FUNCTION_BLOCK GR_plant_Without_NDT
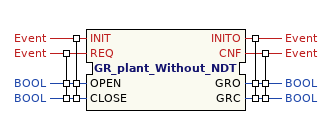
  EVENT_INPUT
    INIT WITH OPEN, CLOSE;
    REQ WITH OPEN, CLOSE;
  END_EVENT
  EVENT_OUTPUT
    INITO WITH GRO, GRC;
    CNF WITH GRO, GRC;
  END_EVENT
  VAR_INPUT
    OPEN : BOOL;
    CLOSE : BOOL;
  END_VAR
  VAR_OUTPUT
    GRO : BOOL;
    GRC : BOOL;
  END_VAR
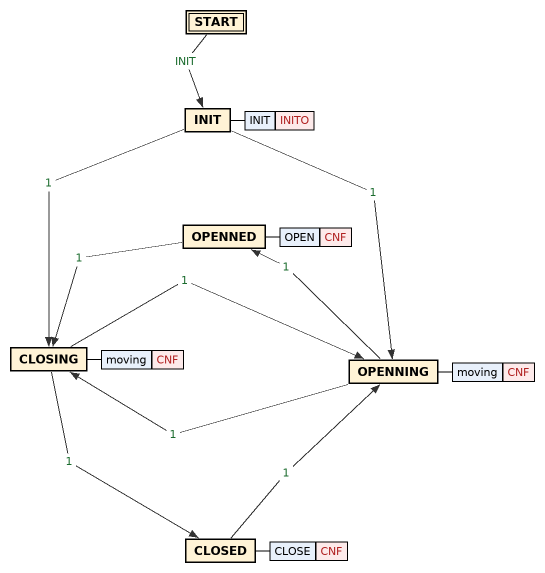
  EC_STATES
    START;
    INIT : INIT -> INITO;
    OPENNED : OPEN -> CNF;
    CLOSED : CLOSE -> CNF;
    OPENNING : moving -> CNF;
    CLOSING : moving -> CNF;
  END_STATES
  EC_TRANSITIONS
    CLOSING TO CLOSED := 1;
    CLOSED TO OPENNING := 1;
    OPENNING TO OPENNED := 1;
    OPENNED TO CLOSING := 1;
    START TO INIT := INIT;
    CLOSING TO OPENNING := 1;
    OPENNING TO CLOSING := 1;
    INIT TO CLOSING := 1;
    INIT TO OPENNING := 1;
  END_TRANSITIONS
  ALGORITHM INIT IN ST:
GRO := FALSE;&#38;#10;GRC := FALSE;&#38;#10;
  END_ALGORITHM
  ALGORITHM OPEN IN ST:
GRO := TRUE;&#38;#10;GRC := FALSE;&#38;#10;
  END_ALGORITHM
  ALGORITHM moving IN ST:
GRO := FALSE;&#38;#10;GRC := FALSE;&#38;#10;
  END_ALGORITHM
  ALGORITHM CLOSE IN ST:
GRC := TRUE;&#38;#10;GRO := FALSE;&#38;#10;
  END_ALGORITHM
  ALGORITHM STOP IN ST:
GRO := FALSE;&#38;#10;GRC := FALSE;&#38;#10;
  END_ALGORITHM
END_FUNCTION_BLOCK
